{attribute 'qualified_only'}
{attribute 'strict'}
TYPE Cylinder :
(
	extend,
	retract
);
END_TYPE

(* stored: Version 1.1.0.1, ProductVersion 3.1.4022.12
   DUT Cylinder: Id {ae6d2e56-4dcc-4582-bbec-31e57f6d7456} *)
